Staubli VAL3: setTool.pgx

public program setTool(num x_nIndexTool)
begin
  // set the TOOL
  jEditPoint.nIndexTool=x_nIndexTool
end
